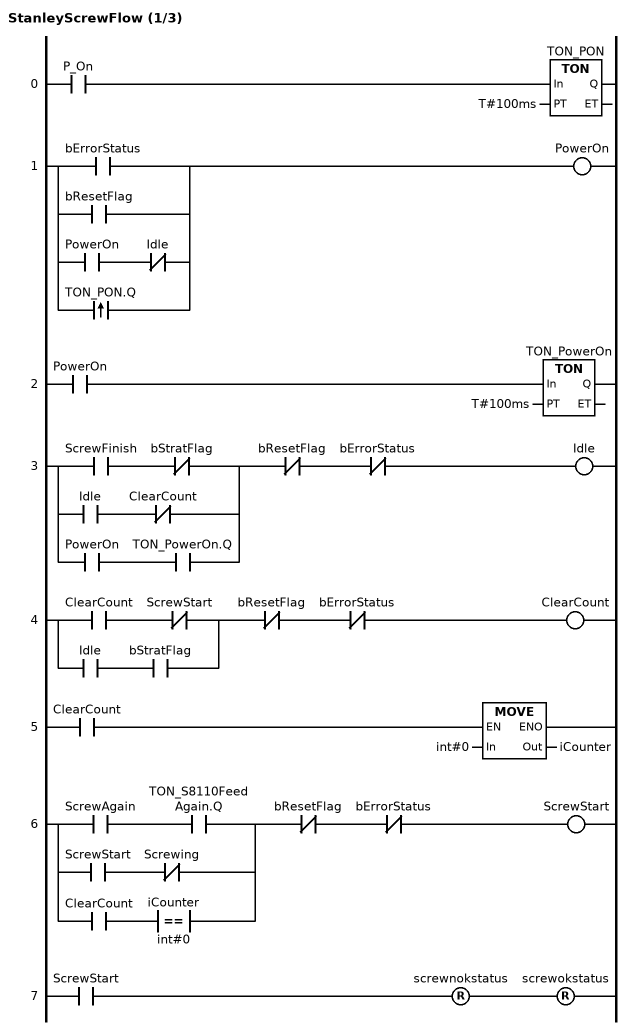
(* [picture p24: StanleyScrewFlow, rungs 0-7] *)
(* Rung 0 *)
TON_PON(In := P_On, PT := T#100ms);
(* Rung 1 *)
_e1(CLK := TON_PON.Q);
PowerOn := bErrorStatus OR bResetFlag OR (PowerOn AND NOT Idle) OR _e1.Q;
(* Rung 2 *)
TON_PowerOn(In := PowerOn, PT := T#100ms);
(* Rung 3 *)
Idle := ((ScrewFinish AND NOT bStratFlag) OR (Idle AND NOT ClearCount) OR (PowerOn AND TON_PowerOn.Q)) AND NOT bResetFlag AND NOT bErrorStatus;
(* Rung 4 *)
ClearCount := ((ClearCount AND NOT ScrewStart) OR (Idle AND bStratFlag)) AND NOT bResetFlag AND NOT bErrorStatus;
(* Rung 5 *)
IF ClearCount THEN iCounter := int#0; END_IF;
(* Rung 6 *)
ScrewStart := ((ScrewAgain AND TON_S8110FeedAgain.Q) OR (ScrewStart AND NOT Screwing) OR (ClearCount AND (iCounter = int#0))) AND NOT bResetFlag AND NOT bErrorStatus;
(* Rung 7 *)
IF ScrewStart THEN
    screwnokstatus := FALSE;
    screwokstatus := FALSE;
END_IF;

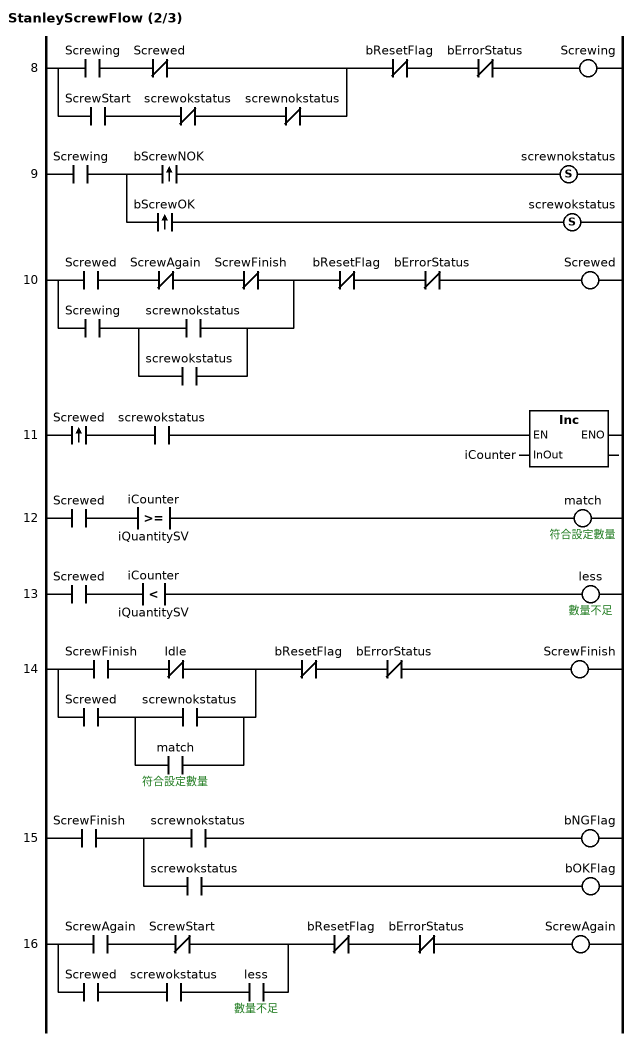
(* Rung 8 *)
Screwing := ((Screwing AND NOT Screwed) OR (ScrewStart AND NOT screwokstatus AND NOT screwnokstatus)) AND NOT bResetFlag AND NOT bErrorStatus;
(* Rung 9 *)
_e2(CLK := bScrewNOK);
IF Screwing AND _e2.Q THEN screwnokstatus := TRUE; END_IF;
_e3(CLK := bScrewOK);
IF Screwing AND _e3.Q THEN screwokstatus := TRUE; END_IF;
(* Rung 10 *)
Screwed := ((Screwed AND NOT ScrewAgain AND NOT ScrewFinish) OR (Screwing AND (screwnokstatus OR screwokstatus))) AND NOT bResetFlag AND NOT bErrorStatus;
(* Rung 11 *)
_e4(CLK := Screwed);
IF _e4.Q AND screwokstatus THEN Inc(InOut := iCounter); END_IF;
(* Rung 12 *)
match := Screwed AND (iCounter >= iQuantitySV);
(* Rung 13 *)
less := Screwed AND (iCounter < iQuantitySV);
(* Rung 14 *)
ScrewFinish := ((ScrewFinish AND NOT Idle) OR (Screwed AND (screwnokstatus OR match))) AND NOT bResetFlag AND NOT bErrorStatus;
(* Rung 15 *)
bNGFlag := ScrewFinish AND screwnokstatus;
bOKFlag := ScrewFinish AND screwokstatus;
(* Rung 16 *)
ScrewAgain := ((ScrewAgain AND NOT ScrewStart) OR (Screwed AND screwokstatus AND less)) AND NOT bResetFlag AND NOT bErrorStatus;

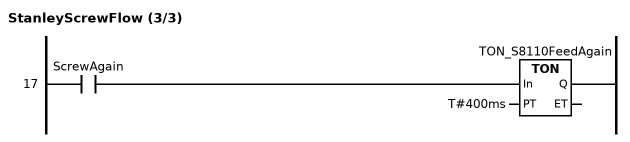
(* Rung 17 *)
TON_S8110FeedAgain(In := ScrewAgain, PT := T#400ms);
END_FUNCTION_BLOCK

FUNCTION_BLOCK StanleyJobSelect
VAR_INPUT
    Enable : BOOL;
    iJobNo : INT;
END_VAR
VAR_OUTPUT
    bJobBit0 : BOOL;
    bJobBit1 : BOOL;
    bJobBit2 : BOOL;
END_VAR
CASE iJobNo OF
    0 : 	bJobBit0:=FALSE;
			bJobBit1 :=FALSE;
			bJobBit2:=FALSE;
			
    1 : 	bJobBit0:=TRUE;
			bJobBit1:=FALSE;
			bJobBit2:=FALSE;
			
    2 : 	bJobBit0:=FALSE;
			bJobBit1:=TRUE;
			bJobBit2:=FALSE;
			
    3 : 	bJobBit0:=TRUE;
			bJobBit1:=TRUE;
			bJobBit2:=FALSE;
			
    4 : 	bJobBit0:=FALSE;
			bJobBit1:=FALSE;
			bJobBit2:=TRUE;
			
    5 : 	bJobBit0:=TRUE;
			bJobBit1:=FALSE;
			bJobBit2:=TRUE;
			
    6 : 	bJobBit0:=FALSE;
			bJobBit1:=TRUE;
			bJobBit2:=TRUE;
			
    7 : 	bJobBit0:=TRUE;
			bJobBit1:=TRUE;
			bJobBit2:=TRUE;
ELSE
    bJobBit0:=FALSE;
	bJobBit1:=FALSE;
	bJobBit2:=FALSE;
END_CASE;
END_FUNCTION_BLOCK

FUNCTION_BLOCK Station_1Step
VAR
    timer_PON : TON;
    PowerOn : BOOL;
    Idle : BOOL;
    Step1Start : BOOL;
    Step1Running : BOOL;
    Step1Finish : BOOL;
END_VAR
VAR_OUTPUT
    outStep1StartFlag : BOOL;
    inoutCurrentStationWork : BOOL;
END_VAR
VAR_INPUT
    Enable : BOOL;
    inAutoStatus : BOOL;
    inResetFlag : BOOL;
    inErrorStatus : BOOL;
    inEnablePB : BOOL;
    inMachineStart : BOOL;
    inExStationFinish : BOOL;
    inExStationOK : BOOL;
    inExStationNG : BOOL;
    inStep1FinishFlag : BOOL;
END_VAR
VAR_IN_OUT
    inoutCurrentStationFinish : BOOL;
    inoutCurrentStationOK : BOOL;
    inoutCurrentStationNG : BOOL;
END_VAR
VAR
    _e1 : R_TRIG;
END_VAR
(* ladder, written here as Structured Text *)

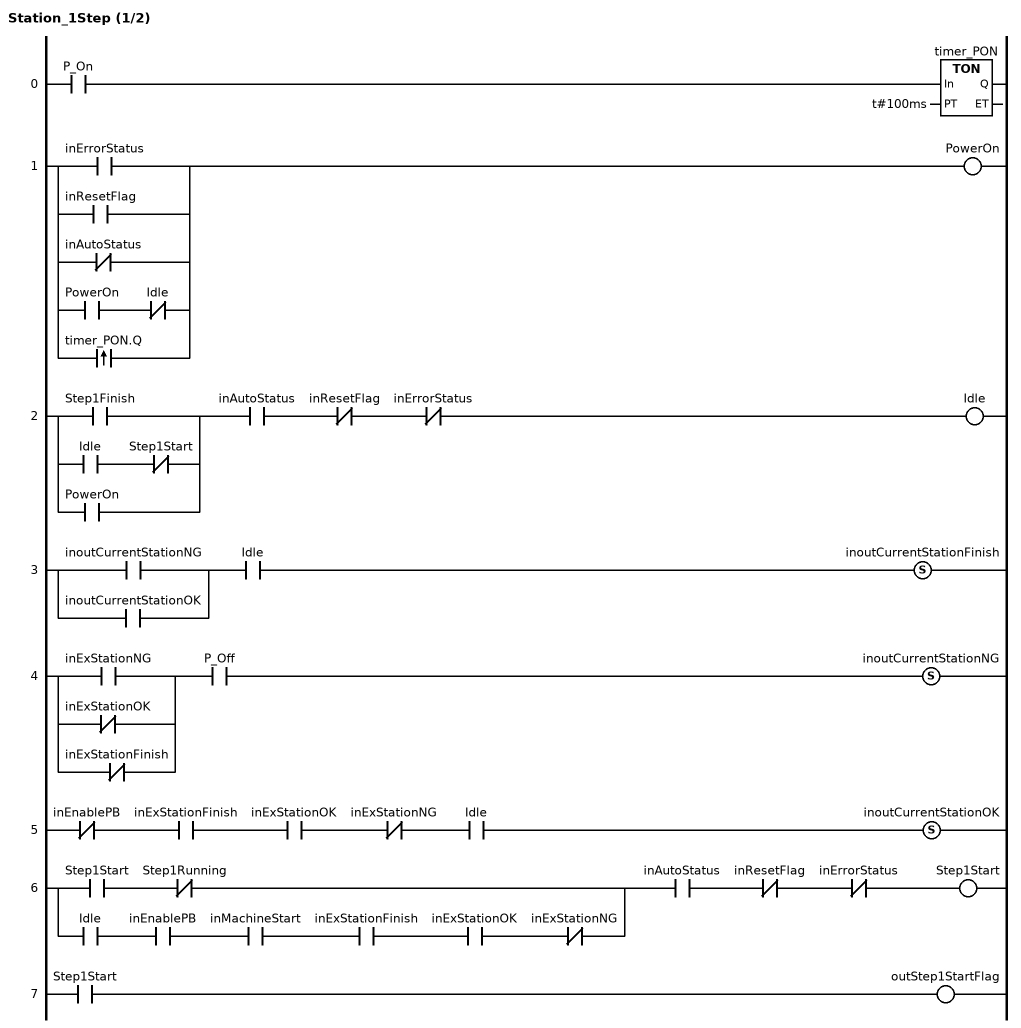
(* Rung 0 *)
timer_PON(In := P_On, PT := t#100ms);
(* Rung 1 *)
_e1(CLK := timer_PON.Q);
PowerOn := inErrorStatus OR inResetFlag OR NOT inAutoStatus OR (PowerOn AND NOT Idle) OR _e1.Q;
(* Rung 2 *)
Idle := (Step1Finish OR (Idle AND NOT Step1Start) OR PowerOn) AND inAutoStatus AND NOT inResetFlag AND NOT inErrorStatus;
(* Rung 3 *)
IF (inoutCurrentStationNG OR inoutCurrentStationOK) AND Idle THEN
    inoutCurrentStationFinish := TRUE;
END_IF;
(* Rung 4 *)
IF (inExStationNG OR NOT inExStationOK OR NOT inExStationFinish) AND P_Off THEN
    inoutCurrentStationNG := TRUE;
END_IF;
(* Rung 5 *)
IF NOT inEnablePB AND inExStationFinish AND inExStationOK AND NOT inExStationNG AND Idle THEN
    inoutCurrentStationOK := TRUE;
END_IF;
(* Rung 6 *)
Step1Start := ((Step1Start AND NOT Step1Running) OR (Idle AND inEnablePB AND inMachineStart AND inExStationFinish AND inExStationOK AND NOT inExStationNG)) AND inAutoStatus AND NOT inResetFlag AND NOT inErrorStatus;
(* Rung 7 *)
outStep1StartFlag := Step1Start;

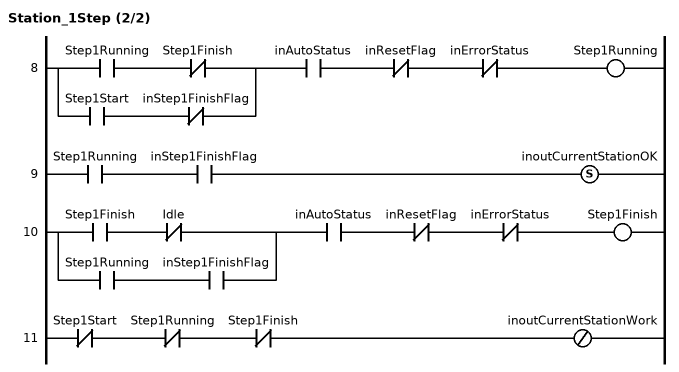
(* Rung 8 *)
Step1Running := ((Step1Running AND NOT Step1Finish) OR (Step1Start AND NOT inStep1FinishFlag)) AND inAutoStatus AND NOT inResetFlag AND NOT inErrorStatus;
(* Rung 9 *)
IF Step1Running AND inStep1FinishFlag THEN inoutCurrentStationOK := TRUE; END_IF;
(* Rung 10 *)
Step1Finish := ((Step1Finish AND NOT Idle) OR (Step1Running AND inStep1FinishFlag)) AND inAutoStatus AND NOT inResetFlag AND NOT inErrorStatus;
(* Rung 11 *)
inoutCurrentStationWork := NOT (NOT Step1Start AND NOT Step1Running AND NOT Step1Finish);
END_FUNCTION_BLOCK

FUNCTION_BLOCK Station_2Step
VAR
    timer_PON : TON;
    PowerOn : BOOL;
    Idle : BOOL;
    Step1Start : BOOL;
    Step1Running : BOOL;
    Step1Finish : BOOL;
    Step2Start : BOOL;
    Step2Running : BOOL;
    Step2Finish : BOOL;
END_VAR
VAR_OUTPUT
    outStep1StartFlag : BOOL;
    outStep2StartFlag : BOOL;
    inoutCurrentStationWork : BOOL;
END_VAR
VAR_INPUT
    Enable : BOOL;
    inAutoStatus : BOOL;
    inResetFlag : BOOL;
    inErrorStatus : BOOL;
    inEnablePB : BOOL;
    inMachineStart : BOOL;
    inExStationFinish : BOOL;
    inExStationOK : BOOL;
    inExStationNG : BOOL;
    inStep1FinishFlag : BOOL;
    inStep2OKFlag : BOOL;
    inStep2NGFlag : BOOL;
END_VAR
VAR_IN_OUT
    inoutCurrentStationFinish : BOOL;
    inoutCurrentStationOK : BOOL;
    inoutCurrentStationNG : BOOL;
END_VAR
VAR
    _e1 : R_TRIG;
END_VAR
(* ladder, written here as Structured Text *)

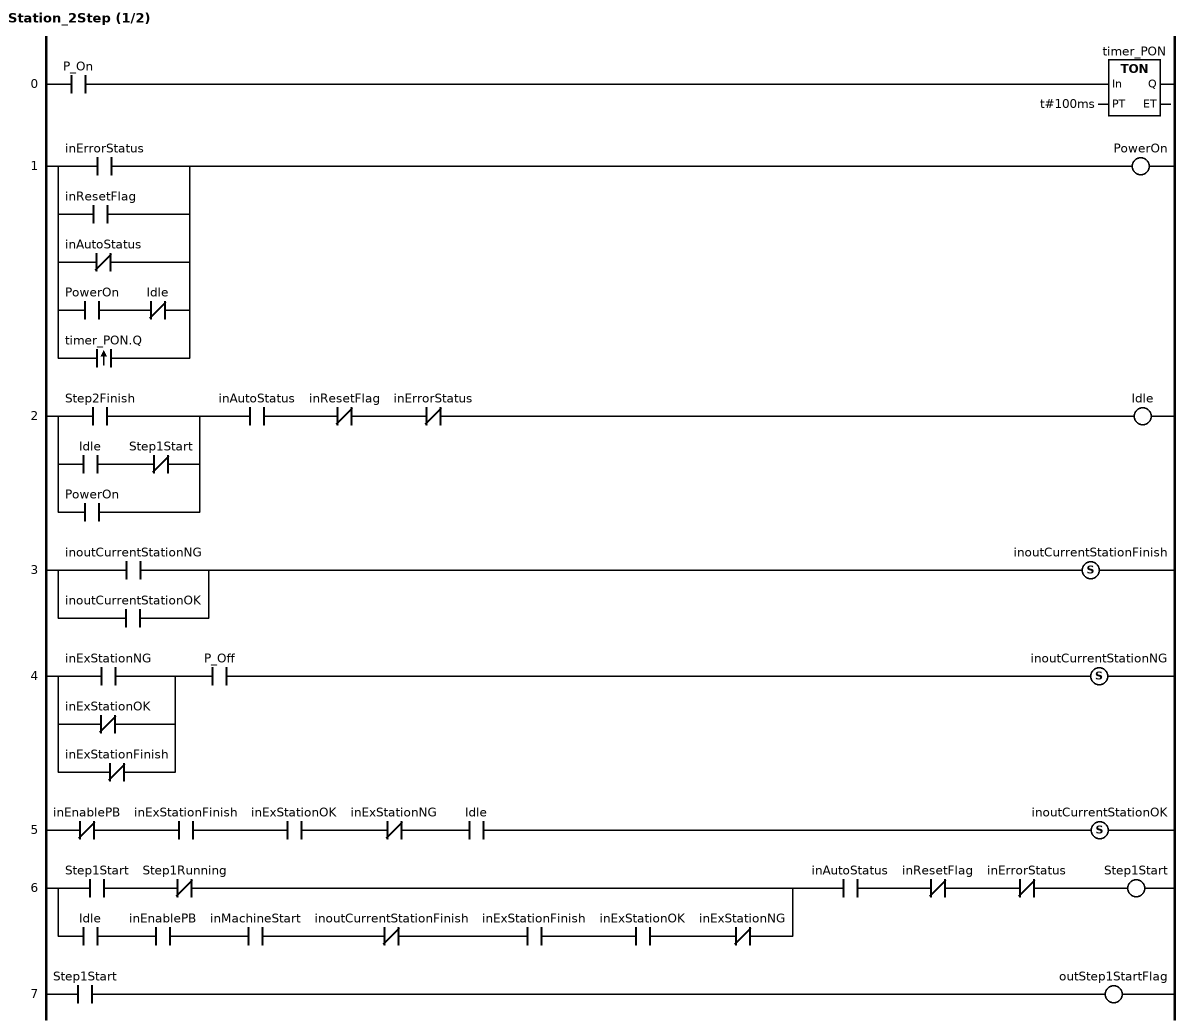
(* Rung 0 *)
timer_PON(In := P_On, PT := t#100ms);
(* Rung 1 *)
_e1(CLK := timer_PON.Q);
PowerOn := inErrorStatus OR inResetFlag OR NOT inAutoStatus OR (PowerOn AND NOT Idle) OR _e1.Q;
(* Rung 2 *)
Idle := (Step2Finish OR (Idle AND NOT Step1Start) OR PowerOn) AND inAutoStatus AND NOT inResetFlag AND NOT inErrorStatus;
(* Rung 3 *)
IF inoutCurrentStationNG OR inoutCurrentStationOK THEN inoutCurrentStationFinish := TRUE; END_IF;
(* Rung 4 *)
IF (inExStationNG OR NOT inExStationOK OR NOT inExStationFinish) AND P_Off THEN
    inoutCurrentStationNG := TRUE;
END_IF;
(* Rung 5 *)
IF NOT inEnablePB AND inExStationFinish AND inExStationOK AND NOT inExStationNG AND Idle THEN
    inoutCurrentStationOK := TRUE;
END_IF;
(* Rung 6 *)
Step1Start := ((Step1Start AND NOT Step1Running) OR (Idle AND inEnablePB AND inMachineStart AND NOT inoutCurrentStationFinish AND inExStationFinish AND inExStationOK AND NOT inExStationNG)) AND inAutoStatus AND NOT inResetFlag AND NOT inErrorStatus;
(* Rung 7 *)
outStep1StartFlag := Step1Start;

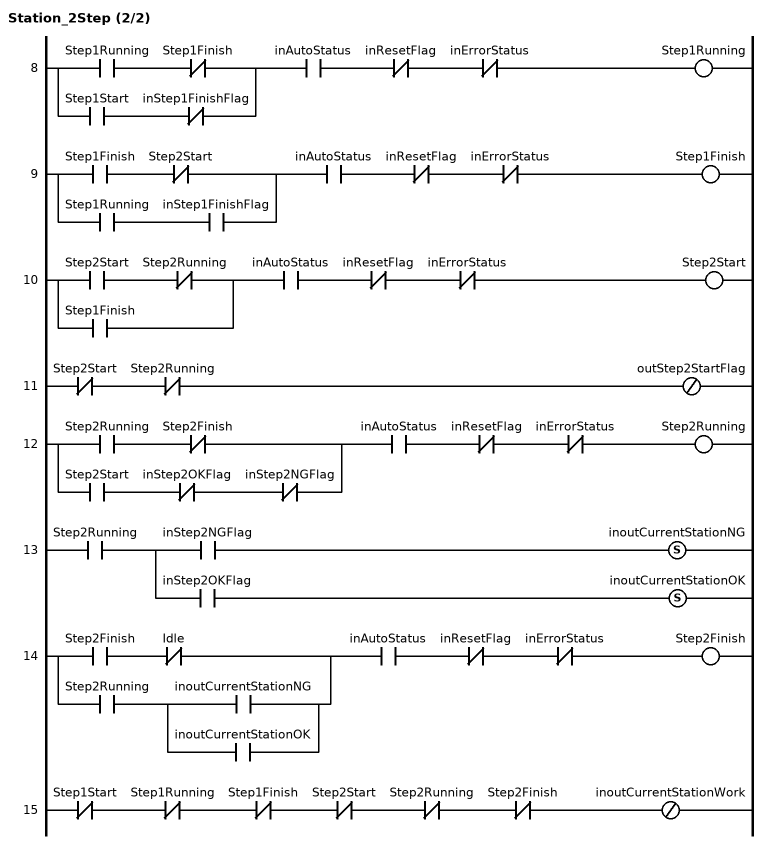
(* Rung 8 *)
Step1Running := ((Step1Running AND NOT Step1Finish) OR (Step1Start AND NOT inStep1FinishFlag)) AND inAutoStatus AND NOT inResetFlag AND NOT inErrorStatus;
(* Rung 9 *)
Step1Finish := ((Step1Finish AND NOT Step2Start) OR (Step1Running AND inStep1FinishFlag)) AND inAutoStatus AND NOT inResetFlag AND NOT inErrorStatus;
(* Rung 10 *)
Step2Start := ((Step2Start AND NOT Step2Running) OR Step1Finish) AND inAutoStatus AND NOT inResetFlag AND NOT inErrorStatus;
(* Rung 11 *)
outStep2StartFlag := NOT (NOT Step2Start AND NOT Step2Running);
(* Rung 12 *)
Step2Running := ((Step2Running AND NOT Step2Finish) OR (Step2Start AND NOT inStep2OKFlag AND NOT inStep2NGFlag)) AND inAutoStatus AND NOT inResetFlag AND NOT inErrorStatus;
(* Rung 13 *)
IF Step2Running AND inStep2NGFlag THEN inoutCurrentStationNG := TRUE; END_IF;
IF Step2Running AND inStep2OKFlag THEN inoutCurrentStationOK := TRUE; END_IF;
(* Rung 14 *)
Step2Finish := ((Step2Finish AND NOT Idle) OR (Step2Running AND (inoutCurrentStationNG OR inoutCurrentStationOK))) AND inAutoStatus AND NOT inResetFlag AND NOT inErrorStatus;
(* Rung 15 *)
inoutCurrentStationWork := NOT (NOT Step1Start AND NOT Step1Running AND NOT Step1Finish AND NOT Step2Start AND NOT Step2Running AND NOT Step2Finish);
END_FUNCTION_BLOCK